# EPICS substitutions: sbtest-mk-iocApp/Db/userHost2.substitutions
# Example substitutions file

#file "db/asub.db" {
#    { user = "mrippaHost" }
#
#}

file db/asub2.db {
    pattern { user, no, scan }
        { "sim2", 2, "Passive" }
}
